FUNCTION_BLOCK E_TRAIN (* Composite Function Block Type *)
  (* Standard: 61499-2 *)
  (* Version 0.0, 9/9/2026, lizar, Schneider Electric, template *)
  PACKAGE Main;
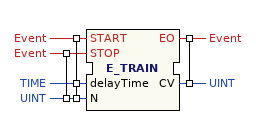
  EVENT_INPUT
    START WITH delayTime, N; (* Initialization Request *)
    STOP WITH N; (* Normal Execution Request *)
  END_EVENT
  EVENT_OUTPUT
    EO WITH CV; (* Initialization Confirm *)
  END_EVENT
  VAR_INPUT
    delayTime : TIME; (* Input event qualifier *)
    N : UINT;
  END_VAR
  VAR_OUTPUT
    CV : UINT; (* Output event qualifier *)
  END_VAR
  FBS
    FB1 : E_CYCLE;
    FB2 : E_CTU;
    FB4 : E_PERMIT;
    FB5 : TWO_I_TWO_O;
    FB3 : E_SPLIT;
  END_FBS
  EVENT_CONNECTIONS
    START TO FB1.START;
    FB4.EO TO FB5.FB5_EI2;
    STOP TO FB5.FB5_EI1;
    FB5.FB6_EO1 TO FB1.STOP;
    FB5.FB6_EO2 TO FB2.R;
    FB2.CUO TO FB4.EI;
    FB1.EO TO FB3.EI;
    FB3.EO1 TO EO;
    FB3.EO2 TO FB2.CU;
  END_CONNECTIONS
  DATA_CONNECTIONS
    N TO FB2.PV;
    delayTime TO FB1.DT;
    FB2.CV TO CV;
    FB2.Q TO FB4.PERMIT;
  END_CONNECTIONS
END_FUNCTION_BLOCK
